Staubli VAL3: ALGORITH.dtx

trsf trCut[100]
num nThickRadio = 100
